TYPE ST_MotionStep :
STRUCT
	fTargetX		: LREAL; // Target position of X axis - AXIS1, X axis kohde asento
	fTargetY		: LREAL; // Target position of Y axis - AXIS2, Y axis kohde asento
	nZaction		: INT; 	 // 1 = Lift, 2 = Lower, 0 = Do nothing, nostimen asennot
END_STRUCT
END_TYPE

(* stored: Version 1.1.0.1, ProductVersion 3.1.4024.12
   DUT ST_MotionStep: Id {c558b0b0-c766-4ec8-962e-e3e446a5acc6} *)
